// TIA Portal V19 export
TYPE "Alarm_Parameter_Wort"
   STRUCT
      Parameter : Array[0..15] of "Alarm_Parameter";
   END_STRUCT;
END_TYPE
